TYPE sWeight :
STRUCT
	pv : LREAL := -10000.0;
	status : string(15) := 'Invalid';
END_STRUCT
END_TYPE

(* stored: Version 1.1.0.1, ProductVersion 3.1.0.36
   DUT sWeight: Id {a3e7cef3-21f6-4110-9f53-6cbcafd2ba42} *)
